// TwinCAT 3 PLC project GarageDoor
// ProgramVersion: 3.1.4024.0
// libraries:
//   CmpBitmapPool, * (System)
//   Tc2_Standard, * (Beckhoff Automation GmbH)
//   Tc2_System, * (Beckhoff Automation GmbH)
//   Tc3_Module, * (Beckhoff Automation GmbH)
// project tree:
//   / GlobalTextList.TcGTLO, PlcTask.TcTTO, Visualization Manager.TcVMO (not stored)
//   POUs/ Blinker.TcPOU, GarageDoor.TcPOU, ImagePool.TcIPO (not stored), MAIN.TcPOU, OpenCloseGarage.TcPOU, Visualization.TcVIS

CONFIGURATION GarageDoor
    RESOURCE PLC ON TwinCAT3
        TASK PlcTask(INTERVAL := T#10ms, PRIORITY := 20);
        PROGRAM MAIN WITH PlcTask : MAIN;
    END_RESOURCE
END_CONFIGURATION

// ---- POUs/MAIN.TcPOU
PROGRAM MAIN
VAR
END_VAR

GarageDoor();

END_PROGRAM

// ---- POUs/GarageDoor.TcPOU
PROGRAM GarageDoor
VAR
	bActuationButton AT %I* : BOOL; //actuation button connected through visualization
	bOpenSensor AT %Q* : BOOL;
	bClosedSensor AT %Q* : BOOL; //sensor conected to lights 
	bDriveOverloadSensor : BOOL; //sensor that indicates if there is an error
	bLightForMotion : BOOL; // light that turns on if the door is in motion
	fbGarage : OpenCloseGarage;
	bVisualizationOpenClose : BOOL;
	bPauseLight AT %Q* : BOOL; //light that blinks if the door is paused
	bErrorButton AT %I* : BOOL; //button that puts the door in error
END_VAR

fbGarage.bActuationProgram := bActuationButton; //we activate the garage

bOpenSensor := fbGarage.bDoorOpen;
bClosedSensor := fbGarage.bDoorClosed;
bDriveOverloadSensor := fbGarage.bDriveOverload; //we set the sensors

bLightForMotion := fbGarage.bLight;
bVisualizationOpenClose := fbGarage.bVisualization;


bPauseLight := fbGarage.bLightForPause;

fbGarage.bError := bErrorButton;



fbGarage();

END_PROGRAM

// ---- POUs/OpenCloseGarage.TcPOU
FUNCTION_BLOCK OpenCloseGarage
VAR_INPUT
	bActuationProgram : BOOL; //the input we give through the interfac
	bError : BOOL; //light that paused the door
END_VAR
VAR_OUTPUT
	bLight : BOOL; //garage light that turns on if the garage is opening or closing (blinks if there is an error or the garage failed to open/close
	bDoorOpen : BOOL; //sensor that indicates wheather or not the garage door is opened
	bDoorClosed : BOOL; //sensor that indicate wheather or not the garage is closed
	bDriveOverload : BOOL; //sensor that indicates if there is an error or if the garage takes too log to open/closLight
	bLightForPause : BOOL;
	bVisualization : BOOL; //bool varable for visual effects
END_VAR
VAR
	iState : UDINT; //states variable which we use to go through states
	fbOpen : TON; //time that opens the door
	fbClose : TON; //timer that closes the door
	fbInitial : R_TRIG; //trigger for setting the initial position of the door to closed
	bInitialActivate : BOOL; //bool variable that activates the initial trigger
	fbBlink : Blinker;
	bActuation : BOOL; //actuation button which closes/opens the door
	
	bTempOp : BOOL; //temp open variable, helps in the error state
	bTempCls : BOOL; //temp closed variable,helps in the error state
	
	fbActivate : R_TRIG; // trigger for activation
END_VAR

bInitialActivate := TRUE; //we close the door at the start
fbInitial(CLK := TRUE);
IF fbInitial.Q THEN
	bDoorClosed := TRUE; //we have set the door to closed at the start (only activates the first time we run the program
END_IF

CASE iState OF
	0:
		fbActivate(CLK := bActuationProgram);
		IF fbActivate.Q THEN
			bActuation := TRUE;
		END_IF
		IF bActuation THEN
			iState := 10; //if we click the button go to the next state and check it's state
		END_IF
	5: //forgot to turn off actuation added an extra state
		bActuation := FALSE;
		iState := 0; //return to the first state	
	10:
		IF bDoorOpen THEN
			bDoorOpen := FALSE;
			iState := 20; //if opened go to state 20
		ELSIF bDoorClosed THEN
			bDoorClosed := FALSE;
			iState := 30; //if closed go to state 30
		ELSIF bDriveOverload THEN
			bDoorClosed := FALSE;
			bDoorOpen := FALSE;
			bActuation := FALSE; //we turn off the actuation button
			iState := 50; //if there is an error go to state 40
		END_IF
	15:
		bActuation := FALSE;
		iState := 50;
	20:	
		fbActivate(CLK := bActuationProgram);
		IF fbActivate.Q THEN
			bActuation := FALSE;
		END_IF	
		IF bError THEN
			iState := 15; //incase the door goes to error
		END_IF
		IF bActuation THEN
			fbClose.IN := TRUE; //we start closing it
			bLight := TRUE; //we turn the light on             
			bTempCls := TRUE; //set the temp to true
			IF fbClose.Q THEN //if it finished closing
				bTempCls := FALSE; //set the temp to false
				bDoorClosed := TRUE; //turn the closed sensor on
				fbClose.IN := FALSE; //reset timer
				bLight := FALSE; //turn the light off
				iState := 5; //turn off actuation
			END_IF
		ELSE
			bLightForPause := TRUE;
			iState := 40; //if we stopped the door go to the pause state
		END_IF

			
	30: //if the door is closed
		fbActivate(CLK := bActuationProgram);
		IF fbActivate.Q THEN
			bActuation := FALSE;
		END_IF
		IF bError THEN
			iState := 15; //incase the door goes to error
		END_IF
		IF bActuation THEN
			fbOpen.IN := TRUE; //we start opening it
			bLight := TRUE; //we turn the light on
			bTempOp := TRUE;// set the temp open to true
			IF fbOpen.Q THEN //if it finished opening
				bTempOp := FALSE;
				bDoorOpen := TRUE; //turn the open sensor on
				fbOpen.IN := FALSE; //reset timer
				bLight := FALSE; //turn the light off
				iState := 5; //turn off actuation
			END_IF
		ELSE
			bLightForPause := TRUE;
			iState := 40; //if we paused the door go to the pause state for open
		END_IF
	40:
		IF bError THEN
			bDriveOverload := TRUE;
			iState := 15; //incase the door goes to error
		END_IF
		bVisualization := TRUE;
		fbOpen.IN := FALSE; //reset the timers
		fbClose.IN := FALSE;
		bDoorClosed := FALSE;
		bDoorOpen := FALSE; //we set the door states to false
		fbActivate(CLK := bActuationProgram);
		IF fbActivate.Q THEN
			bActuation := TRUE;
			bLightForPause := FALSE; //we turn off the pause light
		END_IF
		IF bActuation AND bTempOp THEN //if we press the actuation button and the door was opening
			bLight := TRUE;
			fbClose.IN := TRUE;
			IF fbClose.Q THEN
				bVisualization := FALSE;
				bDoorClosed := TRUE; //we closed the door
 				bLight := FALSE;
				bTempOp := FALSE;
				fbClose.IN := FALSE;
				bDriveOverload := FALSE;
				iState := 5; //turn off actuation
			END_IF	
		END_IF
		IF bActuation AND bTempCls THEN //if we press the actuation button and the door was opening
			bLight := TRUE;
			fbOpen.IN := TRUE;
			IF fbOpen.Q THEN
				bVisualization := FALSE;
				bDoorOpen := TRUE; //we opened the door
 				bLight := FALSE;
				bTempCls := FALSE;
				fbOpen.IN := FALSE;
				bDriveOverload := FALSE;
				iState := 5; //turn actuation off
			END_IF	
		END_IF
				
	50: //error state
		bLight := fbBlink.bBlink; //we mak the light blink
		fbBlink();
		bDriveOverload := TRUE;
		fbOpen.IN := FALSE; //reset the timers
		fbClose.IN := FALSE;
		bDoorClosed := FALSE;
		bDoorOpen := FALSE; //we set the door states to false
		bVisualization := FALSE;
		bLightForPause := FALSE;
		fbActivate(CLK := bActuationProgram);
		IF fbActivate.Q THEN
			bActuation := TRUE;
		END_IF
		IF bActuation AND bTempOp THEN //if we press the actuation button and the door was opening
			bLight := TRUE;
			fbClose.IN := TRUE;
			bDriveOverload := FALSE;
			IF fbClose.Q THEN
				bDoorClosed := TRUE; //we closed the door
 				bLight := FALSE;
				bTempOp := FALSE;
				fbClose.IN := FALSE;
				iState := 5; //turn off actuation
			END_IF	
		END_IF
		IF bActuation AND bTempCls THEN //if we press the actuation button and the door was opening
			bLight := TRUE;
			fbOpen.IN := TRUE;
			bDriveOverload := FALSE;
			IF fbOpen.Q THEN
				bDoorOpen := TRUE; //we opened the door
 				bLight := FALSE;
				bTempCls := FALSE;
				fbOpen.IN := FALSE;
				iState := 5; //turn actuation off
			END_IF	
		END_IF
END_CASE

fbOpen(PT := T#7000MS);
fbClose(PT := T#7000MS);

END_FUNCTION_BLOCK

// ---- POUs/Blinker.TcPOU
FUNCTION_BLOCK Blinker
VAR_INPUT
END_VAR
VAR_OUTPUT
	bBlink : BOOL; //bool variable that sets the light on/off constantly
END_VAR
VAR
	fbTimer1 : TON;
	fbTimer2 : TON;
	fbTimer3 : TON;
	
	iStateFB : INT; //state variable to switch between states in the blinker function block
END_VAR

CASE iStateFB OF
	0:
		bBlink := TRUE;
		fbTimer1.IN := TRUE;
		iStateFB := 10;
	10:	
		IF fbTimer1.Q THEN
			bBlink := FALSE;
			fbTimer1.IN := FALSE;
			fbTimer2.IN := TRUE;
			iStateFB := 20;
		END_IF
	20:
		IF fbTimer2.Q THEN
			bBlink := TRUE;
			fbTimer2.IN := FALSE;
			fbTimer3.IN := TRUE;
			iStateFB := 30;
		END_IF	
	30:
		IF fbTimer3.Q THEN
			bBlink := FALSE;
			fbTimer3.IN := FALSE;
			iStateFB := 0;
		END_IF	
END_CASE

fbTimer1(PT := T#400MS);// timers for blinkers
fbTimer2(PT := T#400MS);
fbTimer3(PT := T#400MS);

END_FUNCTION_BLOCK

// ---- GlobalTextList.TcGTLO
TEXTLIST GlobalTextList
  275 = 'Actuation'
  58 = 'Closed'
  950 = 'Driveoverload'
  807 = 'Error'
  139 = 'Opened'
  127 = 'Pause'
  858 = 'Paused'
  226 = 'THE DOOR HAD AN ERROR PRESS THE ACTUATION BUTTON TO FIX IT'
END_TEXTLIST

// ---- POUs/Visualization.TcVIS
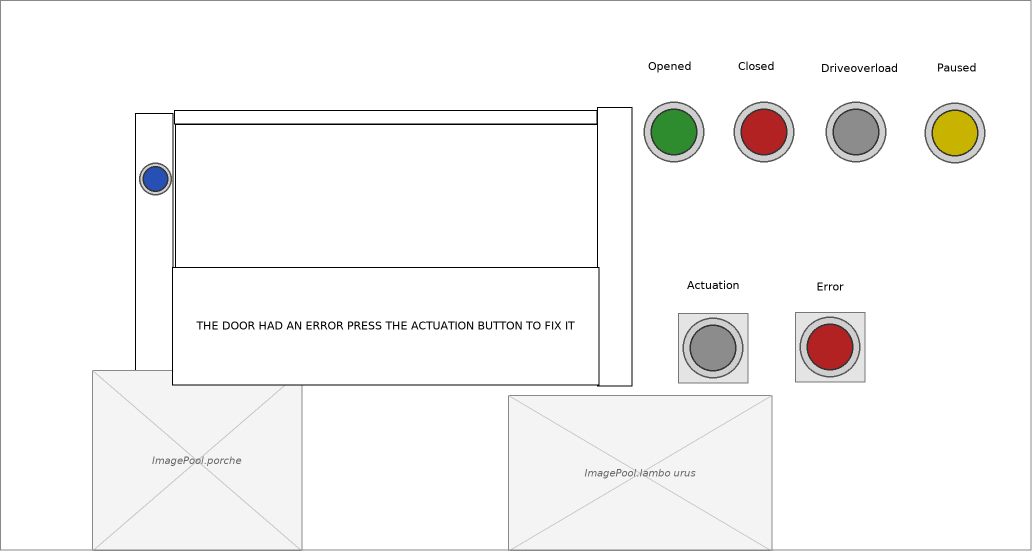
VISUALIZATION Visualization  // 1032x551
    Rectangle (175,124 424x261), invisible if: GarageDoor.bOpenSensor
    Rectangle (135,113 38x274)
    Rectangle (597,107 35x279)
    Rectangle (174,110 423x14)
    Lamp1 (136,160 39x38), variable: GarageDoor.bLightForMotion, style: Lamp-Lamp1-Blue
    Lamp1 (639,97 70x70), variable: GarageDoor.bOpenSensor, style: Lamp-Lamp1-Green
    Lamp1 (729,97 70x70), variable: GarageDoor.bClosedSensor, style: Lamp-Lamp1-Red
    Lamp1 (821,97 70x70), variable: GarageDoor.bDriveOverloadSensor, style: Lamp-Lamp1-Gray
    Label (637,52 66x29), "Opened"
    Label (730,55 53x23), "Closed"
    Label (816,57 87x23), "Driveoverload"
    PushSwitch (678,313 70x70), variable: GarageDoor.bActuationButton, behaviour: TAP, style: Switch-PushSwitch-Gray
    PushSwitch (795,312 70x70), variable: GarageDoor.bErrorButton, behaviour: TAP, style: Switch-PushSwitch-Red
    Label (804,263 52x48), "Error"
    Label (688,268 51x35), "Actuation"
    Lamp1 (920,98 70x70), variable: GarageDoor.bPauseLight, style: Lamp-Lamp1-Yellow
    Label (882,53 150x30), "Paused"
    Image (92,370 210x181), image: ImagePool.porche
    Image (508,395 264x156), image: ImagePool.lambo urus
    Rectangle (175,267 422x118), invisible if: NOT GarageDoor.bVisualizationOpenClose
    Rectangle (172,267 427x118), "THE DOOR HAD AN ERROR PRESS THE ACTUATION BUTTON TO FIX IT", invisible if: NOT GarageDoor.bDriveOverloadSensor
END_VISUALIZATION
